(* PLC project 06_move_add.project, CODESYS CODESYS V3.5 SP22 Patch 2 *)
(* stored: creationDateTime 2026-07-24T04:57:24.5952907, modificationDateTime 2026-07-24T04:57:07.7288124 *)

PROGRAM PLC_PRG
  VAR
    xEnable : BOOL;
    xMoveExecuted : BOOL;
    xAddExecuted : BOOL;
    nSource : DINT;
    nDestination : DINT;
    nIncrement : DINT := 1;
  END_VAR

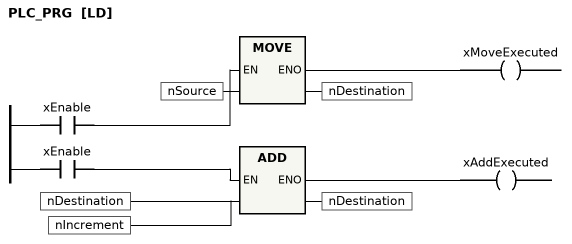
(* LD diagram, written out as Structured Text *)

IF xEnable THEN nDestination := nSource; END_IF;
xMoveExecuted := xEnable;

IF xEnable THEN nDestination := nDestination + nIncrement; END_IF;
xAddExecuted := xEnable;
END_PROGRAM

CONFIGURATION Application
  RESOURCE Application ON PLC
    TASK MainTask(INTERVAL := T#20ms, PRIORITY := 1);
    PROGRAM PLC_PRG WITH MainTask : PLC_PRG;
  END_RESOURCE
END_CONFIGURATION
